// TIA Portal V20 export
TYPE "GetDiag"
// stored: Access Published, Namespace LineD1
   STRUCT
      DiagMode : UInt := 1;
      CommID : HW_ANY;
      ReturnValue : Int;
      CountDiagDetail : UInt;
      MyDiag : DIS;
   END_STRUCT;
END_TYPE
